Staubli VAL3: split.pgx

program split(string x_sText (dimensions=1), string x_sSep (dimensions=1), string& x_sResult[] (dimensions=1))
  local num i
  local num n
begin
  i=0
  do
    n=find(x_sText,x_sSep)
    if n>0
      x_sResult[i]=left(x_sText,n)
      x_sText=right(x_sText,len(x_sText)-(n+1))
      i=i+1
    endIf
  until n==-1
  x_sResult[i]=x_sText
end
